{attribute 'qualified_only'}
{attribute 'strict'}
TYPE E_RS_BASE_READ_TYPE :
(
	SINGLE			:= 0,
	SINGLE_USER,
	PERIODIC,
	PERIODIC_USER
);
END_TYPE

(* stored: Version 1.1.0.1, ProductVersion 3.1.4022.16
   DUT E_RS_BASE_READ_TYPE: Id {a50598b0-5e20-44f2-8d26-3f64391efa7a} *)
